// TIA Portal V21 export
VAR_GLOBAL   // PLC tag table "DIAG"
   D_Supply_MOD2 AT %I200.0 : Bool;   //    {ExternalWritable false}
   D_Supply_MOD3 AT %I200.1 : Bool;   //    {ExternalWritable false}
   D_Supply_MOD4 AT %I200.2 : Bool;   //    {ExternalWritable false}
   D_Supply_MOD5 AT %I200.3 : Bool;   //    {ExternalWritable false}
   D_Reserve_200_4 AT %I200.4 : Bool;   //    {ExternalWritable false}
   D_Reserve_200_5 AT %I200.5 : Bool;   //    {ExternalWritable false}
   D_Reserve_200_6 AT %I200.6 : Bool;   //    {ExternalWritable false}
   D_Reserve_200_7 AT %I200.7 : Bool;   //    {ExternalWritable false}
   D_Reserve_201_0 AT %I201.0 : Bool;   //    {ExternalWritable false}
   D_Reserve_201_1 AT %I201.1 : Bool;   //    {ExternalWritable false}
   D_Reserve_201_2 AT %I201.2 : Bool;   //    {ExternalWritable false}
   D_Reserve_201_3 AT %I201.3 : Bool;   //    {ExternalWritable false}
   D_Reserve_201_4 AT %I201.4 : Bool;   //    {ExternalWritable false}
   D_Reserve_201_5 AT %I201.5 : Bool;   //    {ExternalWritable false}
   D_Reserve_201_6 AT %I201.6 : Bool;   //    {ExternalWritable false}
   D_Reserve_201_7 AT %I201.7 : Bool;   //    {ExternalWritable false}
   D_Reserve_202_0 AT %I202.0 : Bool;   //    {ExternalWritable false}
   D_Reserve_202_1 AT %I202.1 : Bool;   //    {ExternalWritable false}
   D_Reserve_202_2 AT %I202.2 : Bool;   //    {ExternalWritable false}
   D_Reserve_202_3 AT %I202.3 : Bool;   //    {ExternalWritable false}
   D_Reserve_202_4 AT %I202.4 : Bool;   //    {ExternalWritable false}
   D_Reserve_202_5 AT %I202.5 : Bool;   //    {ExternalWritable false}
   D_Reserve_202_6 AT %I202.6 : Bool;   //    {ExternalWritable false}
   D_Reserve_202_7 AT %I202.7 : Bool;   //    {ExternalWritable false}
   D_Reserve_203_0 AT %I203.0 : Bool;   //    {ExternalWritable false}
   D_Reserve_203_1 AT %I203.1 : Bool;   //    {ExternalWritable false}
   D_Reserve_203_2 AT %I203.2 : Bool;   //    {ExternalWritable false}
   D_Reserve_203_3 AT %I203.3 : Bool;   //    {ExternalWritable false}
   D_Reserve_203_4 AT %I203.4 : Bool;   //    {ExternalWritable false}
   D_Reserve_203_5 AT %I203.5 : Bool;   //    {ExternalWritable false}
   D_Reserve_203_6 AT %I203.6 : Bool;   //    {ExternalWritable false}
   D_Reserve_203_7 AT %I203.7 : Bool;   //    {ExternalWritable false}
   D_Feedback_MOD2 AT %I204.0 : Bool;   //    {ExternalWritable false}
   D_Feedback_MOD3 AT %I204.1 : Bool;   //    {ExternalWritable false}
   D_Feedback_MOD4 AT %I204.2 : Bool;   //    {ExternalWritable false}
   D_Feedback_MOD5 AT %I204.3 : Bool;   //    {ExternalWritable false}
   D_Reserve_204_4 AT %I204.4 : Bool;   //    {ExternalWritable false}
   D_Reserve_204_5 AT %I204.5 : Bool;   //    {ExternalWritable false}
   D_Reserve_204_6 AT %I204.6 : Bool;   //    {ExternalWritable false}
   D_Reserve_204_7 AT %I204.7 : Bool;   //    {ExternalWritable false}
   D_Reserve_205_0 AT %I205.0 : Bool;   //    {ExternalWritable false}
   D_Reserve_205_1 AT %I205.1 : Bool;   //    {ExternalWritable false}
   D_Reserve_205_2 AT %I205.2 : Bool;   //    {ExternalWritable false}
   D_Reserve_205_3 AT %I205.3 : Bool;   //    {ExternalWritable false}
   D_Reserve_205_4 AT %I205.4 : Bool;   //    {ExternalWritable false}
   D_Reserve_205_5 AT %I205.5 : Bool;   //    {ExternalWritable false}
   D_Reserve_205_6 AT %I205.6 : Bool;   //    {ExternalWritable false}
   D_Reserve_205_7 AT %I205.7 : Bool;   //    {ExternalWritable false}
END_VAR
